PROGRAM MAIN
VAR
	
	running				:	BOOL	:= FALSE;
	packagingMachine	:	PackagingMachine;
	input				:	BOOL;
	
END_VAR

// ready when packagingmachine is initialized
// initialized when in stopped state and modemanager enabled
IF NOT running THEN
	IF machineConfig() THEN
		running := TRUE;
	ELSE
		// configurationError
	END_IF
	
ELSE
	CASE packagingMachine.getSignal() OF
		noSignal:
			packagingMachine();
			
		startSignal:
			packagingMachine.setState(command:=ePMLCommand_Start);
			
		stopSignal:
			packagingMachine.setState(command:=ePMLCommand_Stop);
		
		abortSignal:
			packagingMachine.setState(command:=ePMLCommand_Abort);
				
		resetSignal:
			packagingMachine.setState(command:=ePMLCommand_Reset);
			
		clearSignal:
			packagingMachine.setState(command:=ePMLCommand_Clear);

		productionModeSignal:
			packagingMachine.setMode(modeCommand:=ePMLProtUnitMode_Production);
			
		maintenanceModeSignal:
			packagingMachine.setMode(modeCommand:=ePMLProtUnitMode_Maintenance);
			
		manualModeSignal:
			packagingMachine.setMode(modeCommand:=ePMLProtUnitMode_Manual);
			
	END_CASE
	
END_IF

// machine config is used to initialize all units.

METHOD machineConfig : BOOL
VAR_INPUT
END_VAR
VAR
	initMode		:	E_PMLProtectedUnitMode	:= 	ePMLProtUnitMode_Production;
	initCommand		:	E_PMLCommand			:=	ePMLCommand_Stop;
	
	subUnits	:	ARRAY[1..CONST_GV.nSubUnits] OF UnitBaseClass;
	staubli		:	Robot;
END_VAR

// 		subUnit1 - Staubli
subUnits[1] := staubli;


// 		subUnit2 ... subUnitn
// subUnits[2] := subUnit2;


// initialize
packagingMachine.initialize(arg1	:=	initMode, 
							arg2	:=	initCommand, 
							arg3	:=	ADR(subUnits));

							
// return initialization status							
machineConfig := packagingMachine.initialized;
END_METHOD

END_PROGRAM

(* stored: Version 1.1.0.1, ProductVersion 3.1.4022.16
   POU MAIN: Id {2a1917db-94f7-4612-a0b0-dd24ef0b93ab}, SpecialFunc None
   Method machineConfig: Id {ee0c57fb-4377-4f15-bbe7-651c309e3778} *)
